Fanuc KAREL source: kb00003.KL

-- PROVISIONAL review KL for V770-1; original PC SHA256 00904de4465977e374fcf6c2ece066fcb4604d74ccffc480934571cf868cee0c
-- Incomplete behavior may be omitted. Consult companion uncertainty JSON. Do not deploy.
PROGRAM KB00003
%NOLOCKGROUP
VAR
  P1 : REAL
  RESULT : REAL
BEGIN
  -- UNRESOLVED_PC offsets 5-16; opcodes 2E,23
  -- UNRESOLVED_PC offsets 21-36; opcodes 27,22,76,23
  -- UNRESOLVED_PC offsets 41-45; opcodes 7F
END KB00003
